// TIA Portal V19 export
TYPE "typeSimStates"
   STRUCT
      States : Struct
         State11 : UInt;   // Machine 1 / State 1
         State12 : UInt;   // Machine 1 / State 2
         State13 : UInt;   // Machine 1 / State 3
         State14 : UInt;   // Machine 1 / State 4
         State21 : UInt;   // Machine 2 / State 1
         State22 : UInt;   // Machine 2 / State 2
         State23 : UInt;   // Machine 2 / State 3
         State24 : UInt;   // Machine 2 / State 4
      END_STRUCT;
   END_STRUCT;
END_TYPE
